TYPE T_FileLc_SysDebugInfo :
STRUCT
		udiLogCounter : UDINT;
		uinGetHandleCalls : UINT;
END_STRUCT
END_TYPE

(* stored: Version 1.1.0.1, ProductVersion 3.1.0.25
   DUT T_FileLc_SysDebugInfo: Id {afc088f8-7d5f-40bc-a4fe-ebf8bfcf296c} *)
